{attribute 'qualified_only'}
{attribute 'strict'}
TYPE eStati :
(
	S0 := 0, S1, S2, S3, SE, SA
);
END_TYPE

(* stored: Version 1.1.0.1
   EnumerationTextList eStati: Id {138d00d9-506a-0917-09a7-405fa75e3eab} *)
